// TIA Portal project "station 1 twin" (V17)

(* hardware
DEVICE "S7-1500/ET200MP station_1"  S7-1500 station
   slot 0: "Rail_0"  Rack  6ES7 590-1***0-0AA0
   slot 1: "PLC_1"  CPU 1511C-1 PN  6ES7 511-1CK00-0AB0  V2.5
      slot 3: "CPU display_1"  6ES7591-1AA00-0AA0
      slot 32768: "PROFINET interface_1"  X1
         slot 32769: "Port_1"  X1 P1
         slot 32770: "Port_2"  X1 P2
*)

// ===== PLC "PLC_1"  CPU 1511C-1 PN =====

VAR_GLOBAL   // PLC tag table "Default tag table"
   "program run" AT %M0.0 : Bool;
END_VAR

DATA_BLOCK "NX"   // DB1
{ S7_Optimized_Access := 'TRUE' }
VERSION : 0.1
   VAR
      Start : Bool;
      Stop : Bool;
      Cylinder : Bool;
      Fully_extended : Bool;
      Fully_retracted : Bool;
   END_VAR
BEGIN
END_DATA_BLOCK

ORGANIZATION_BLOCK "Main"   // OB1, LAD, ProgramCycle
TITLE = "Main Program Sweep (Cycle)"
{ S7_Optimized_Access := 'TRUE' }
VERSION : 0.1
   VAR_INPUT
      Initial_Call : Bool;   // Initial call of this OB
      Remanence : Bool;   // =True, if remanent data are available
   END_VAR
BEGIN

REGION Network 1
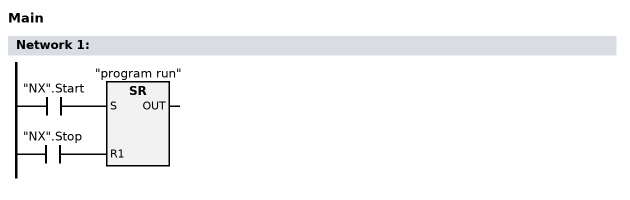
   RUNG wire#powerrail
      Contact( "NX".Start )
      S_SR(operand := "program run", r1 := wire#w1)
   END_RUNG
   RUNG wire#powerrail
      Contact( "NX".Stop )
   END_RUNG wire#w1
   // the same network as SCL:
   IF "NX".Start THEN
       "program run" := TRUE;   // SR flip-flop
   END_IF;
   IF "NX".Stop THEN "program run" := FALSE; END_IF;
END_REGION
END_ORGANIZATION_BLOCK